// TwinCAT 3 PLC project XYZ
// ProgramVersion: 3.1.4024.0
// libraries:
//   Tc2_MC2, * (Beckhoff Automation GmbH)
//   Tc2_Standard, * (Beckhoff Automation GmbH)
//   Tc2_System, * (Beckhoff Automation GmbH)
//   Tc3_MC2_AdvancedHoming, * (Beckhoff Automation GmbH)
//   Tc3_Module, * (Beckhoff Automation GmbH)
//   Tc3_PLCopen_OpcUa, * (Beckhoff Automation GmbH)
// project tree:
//   GVLs/ GlobalSettings.TcGVL
//   / PlcTask.TcTTO
//   POUs/ FB_StorageController.TcPOU, MAIN.TcPOU, PRG_WRITE.TcPOU
// real-time tasks:
//   TASK PlcTask: cycle T#10ms, priority 20, ADS port 350
//   TASK Device 1 (OPC UA Virtual)_Task_58: cycle T#40ms, priority 58, ADS port 351
// motion (NC):
//   TASK NC-Task 1 SAF: cycle T#2ms, priority 4, ADS port 501
//   TASK NC-Task 1 SVB: cycle T#10ms, priority 8, ADS port 511
//   AXIS X1 (id 1)
//     Dynamic: Acceleration=600, Deceleration=600, Jerk=360
//     OtherSettings: AllowMotionCmdToSlave=true
//     encoder EncType=4
//       EncPara: ScaleFactorNumerator=40, ScaleFactorDenominator=12800, Inverse=true, MaxCount=#x0000ffff
//         Inc: RefSearchInverse=true, RefSyncInverse=false, RefMode=1, RefSoftSyncMask=#x0000ffff
//     drive DrvType=24
//       DrvPara: Inverse=true
//         Analog: VeloReferenz=400, ScaleFactorActTorque=0.1
//         TimeComp: TaskDelayCycles=1
//     controller CtrType=1
//       CtrPara: PriorControlFactor=1
//         Observer: BandWidth=20
//   AXIS X2 (id 2)
//     Dynamic: Acceleration=600, Deceleration=600, Jerk=360
//     OtherSettings: AllowMotionCmdToSlave=true
//     encoder EncType=4
//       EncPara: ScaleFactorNumerator=40, ScaleFactorDenominator=12800, Inverse=true, MaxCount=#x0000ffff
//         Inc: RefSearchInverse=true, RefSyncInverse=false, RefMode=1, RefSoftSyncMask=#x0000ffff
//     drive DrvType=24
//       DrvPara: Inverse=true
//         Analog: VeloReferenz=400, ScaleFactorActTorque=0.1
//         TimeComp: TaskDelayCycles=1
//     controller CtrType=1
//       CtrPara: PriorControlFactor=1
//         Observer: BandWidth=20
//   AXIS Z (id 3)
//     Dynamic: Acceleration=1.5, Deceleration=1.5, Jerk=4.5
//     Velo: Maximum=1
//     OtherSettings: AllowMotionCmdToSlave=true
//     encoder EncType=4
//       EncPara: ScaleFactorNumerator=1, ScaleFactorDenominator=12800, MaxCount=#x0000ffff
//         Inc: RefSearchInverse=true, RefSyncInverse=false, RefMode=1, RefSoftSyncMask=#x0000ffff
//     drive DrvType=24
//       Analog: VeloReferenz=1, ScaleFactorActTorque=0.1
//       TimeComp: TaskDelayCycles=1
//     controller CtrType=1
//       CtrPara: PriorControlFactor=1
//         PID: PosKp=1.5
//         Observer: BandWidth=20
//   AXIS Y (id 4)
//     OtherSettings: AllowMotionCmdToSlave=true
//     encoder EncType=4
//       EncPara: ScaleFactorNumerator=40, ScaleFactorDenominator=12800, Inverse=true, MaxCount=#x0000ffff
//         Inc: RefSearchInverse=true, RefSyncInverse=false, RefMode=1, RefSoftSyncMask=#x0000ffff
//     drive DrvType=24
//       DrvPara: Inverse=true
//         Analog: VeloReferenz=400, ScaleFactorActTorque=0.1
//         TimeComp: TaskDelayCycles=1
//     controller CtrType=1
//       CtrPara: PriorControlFactor=1
//         Observer: BandWidth=20
// I/O:
//   DEVICE Device 3 (EtherCAT) (disabled), AmsNetId 192.168.1.197.4.1
//     Term 1 (EK1100) [EK1100 EtherCAT Coupler (2A E-Bus)]
//       Term 2 (EL7031-0030) [EL7031-0030 1Ch. Stepper motor output stage (24V, 2.8A)]
//       Term 3 (EL7031-0030) [EL7031-0030 1Ch. Stepper motor output stage (24V, 2.8A)]
//       Term 4 (EL7031-0030) [EL7031-0030 1Ch. Stepper motor output stage (24V, 2.8A)]
//       Term 5 (EL7031-0030) [EL7031-0030 1Ch. Stepper motor output stage (24V, 2.8A)]
//       Term 6 (EL1008) [EL1008 8Ch. Dig. Input 24V, 3ms]
//       Term 7 (EK1110) [EK1110 EtherCAT extension]
//   DEVICE Device 1 (OPC UA Virtual), AmsNetId 192.168.1.197.2.1
// variable links:
//   NC-Task 1 SAF/Axes/X1 <-> Device 3 (EtherCAT)/Term 1 (EK1100)/Term 2 (EL7031-0030)
//     Drive/Inputs/In/nState1 @bit 3 <-> STM Status/Status/Error
//     Drive/Inputs/In/nState1 @bit 5 <-> STM Status/Status/Moving negative
//     Drive/Inputs/In/nState1 @bit 4 <-> STM Status/Status/Moving positive
//     Drive/Inputs/In/nState1 @bit 1 <-> STM Status/Status/Ready
//     Drive/Inputs/In/nState1 <-> STM Status/Status/Ready to enable
//     Drive/Inputs/In/nState1 @bit 6 <-> STM Status/Status/Torque reduced
//     Drive/Inputs/In/nState1 @bit 2 <-> STM Status/Status/Warning
//     Drive/Inputs/In/nState2 @bit 3 <-> STM Status/Status/Digital input 1
//     Drive/Inputs/In/nState2 @bit 4 <-> STM Status/Status/Digital input 2
//     Drive/Inputs/In/nState2 @bit 5 <-> STM Status/Status/Sync error
//     Drive/Inputs/In/nState2 @bit 7 <-> STM Status/Status/TxPDO Toggle
//     Drive/Inputs/In/nState4 @bit 1 <-> WcState/InputToggle
//     Drive/Inputs/In/nState4 <-> WcState/WcState
//     Drive/Outputs/Out/nCtrl1 <-> STM Control/Control/Enable
//     Drive/Outputs/Out/nCtrl1 @bit 2 <-> STM Control/Control/Reduce torque
//     Drive/Outputs/Out/nCtrl1 @bit 1 <-> STM Control/Control/Reset
//     Drive/Outputs/Out/nDataOut2[0] <-> STM Velocity/Velocity
//     Enc/Inputs/In/nDataIn1[0] <-> ENC Status compact/Counter value
//     Enc/Inputs/In/nDataIn2[0] <-> ENC Status compact/Latch value
//     Enc/Inputs/In/nState1 @bit 4 <-> ENC Status compact/Status/Counter overflow
//     Enc/Inputs/In/nState1 @bit 3 <-> ENC Status compact/Status/Counter underflow
//     Enc/Inputs/In/nState1 @bit 1 <-> ENC Status compact/Status/Latch extern valid
//     Enc/Inputs/In/nState1 @bit 2 <-> ENC Status compact/Status/Set counter done
//     Enc/Inputs/In/nState2 @bit 4 <-> ENC Status compact/Status/Status of extern latch
//     Enc/Inputs/In/nState2 @bit 5 <-> ENC Status compact/Status/Sync error
//     Enc/Inputs/In/nState2 @bit 7 <-> ENC Status compact/Status/TxPDO Toggle
//     Enc/Inputs/In/nState4 @bit 1 <-> WcState/InputToggle
//     Enc/Inputs/In/nState4 <-> WcState/WcState
//     Enc/Outputs/Out/nCtrl1 @bit 3 <-> ENC Control compact/Control/Enable latch extern on negative edge
//     Enc/Outputs/Out/nCtrl1 @bit 1 <-> ENC Control compact/Control/Enable latch extern on positive edge
//     Enc/Outputs/Out/nCtrl1 @bit 2 <-> ENC Control compact/Control/Set counter
//     Enc/Outputs/Out/nDataOut1[0] <-> ENC Control compact/Set counter value
//   NC-Task 1 SAF/Axes/X2 <-> Device 3 (EtherCAT)/Term 1 (EK1100)/Term 3 (EL7031-0030)
//     Drive/Inputs/In/nState1 @bit 3 <-> STM Status/Status/Error
//     Drive/Inputs/In/nState1 @bit 5 <-> STM Status/Status/Moving negative
//     Drive/Inputs/In/nState1 @bit 4 <-> STM Status/Status/Moving positive
//     Drive/Inputs/In/nState1 @bit 1 <-> STM Status/Status/Ready
//     Drive/Inputs/In/nState1 <-> STM Status/Status/Ready to enable
//     Drive/Inputs/In/nState1 @bit 6 <-> STM Status/Status/Torque reduced
//     Drive/Inputs/In/nState1 @bit 2 <-> STM Status/Status/Warning
//     Drive/Inputs/In/nState2 @bit 3 <-> STM Status/Status/Digital input 1
//     Drive/Inputs/In/nState2 @bit 4 <-> STM Status/Status/Digital input 2
//     Drive/Inputs/In/nState2 @bit 5 <-> STM Status/Status/Sync error
//     Drive/Inputs/In/nState2 @bit 7 <-> STM Status/Status/TxPDO Toggle
//     Drive/Inputs/In/nState4 @bit 1 <-> WcState/InputToggle
//     Drive/Inputs/In/nState4 <-> WcState/WcState
//     Drive/Outputs/Out/nCtrl1 <-> STM Control/Control/Enable
//     Drive/Outputs/Out/nCtrl1 @bit 2 <-> STM Control/Control/Reduce torque
//     Drive/Outputs/Out/nCtrl1 @bit 1 <-> STM Control/Control/Reset
//     Drive/Outputs/Out/nDataOut2[0] <-> STM Velocity/Velocity
//     Enc/Inputs/In/nDataIn1[0] <-> ENC Status compact/Counter value
//     Enc/Inputs/In/nDataIn2[0] <-> ENC Status compact/Latch value
//     Enc/Inputs/In/nState1 @bit 4 <-> ENC Status compact/Status/Counter overflow
//     Enc/Inputs/In/nState1 @bit 3 <-> ENC Status compact/Status/Counter underflow
//     Enc/Inputs/In/nState1 @bit 1 <-> ENC Status compact/Status/Latch extern valid
//     Enc/Inputs/In/nState1 @bit 2 <-> ENC Status compact/Status/Set counter done
//     Enc/Inputs/In/nState2 @bit 4 <-> ENC Status compact/Status/Status of extern latch
//     Enc/Inputs/In/nState2 @bit 5 <-> ENC Status compact/Status/Sync error
//     Enc/Inputs/In/nState2 @bit 7 <-> ENC Status compact/Status/TxPDO Toggle
//     Enc/Inputs/In/nState4 @bit 1 <-> WcState/InputToggle
//     Enc/Inputs/In/nState4 <-> WcState/WcState
//     Enc/Outputs/Out/nCtrl1 @bit 3 <-> ENC Control compact/Control/Enable latch extern on negative edge
//     Enc/Outputs/Out/nCtrl1 @bit 1 <-> ENC Control compact/Control/Enable latch extern on positive edge
//     Enc/Outputs/Out/nCtrl1 @bit 2 <-> ENC Control compact/Control/Set counter
//     Enc/Outputs/Out/nDataOut1[0] <-> ENC Control compact/Set counter value
//   NC-Task 1 SAF/Axes/Y <-> Device 3 (EtherCAT)/Term 1 (EK1100)/Term 5 (EL7031-0030)
//     Drive/Inputs/In/nState1 @bit 3 <-> STM Status/Status/Error
//     Drive/Inputs/In/nState1 @bit 5 <-> STM Status/Status/Moving negative
//     Drive/Inputs/In/nState1 @bit 4 <-> STM Status/Status/Moving positive
//     Drive/Inputs/In/nState1 @bit 1 <-> STM Status/Status/Ready
//     Drive/Inputs/In/nState1 <-> STM Status/Status/Ready to enable
//     Drive/Inputs/In/nState1 @bit 6 <-> STM Status/Status/Torque reduced
//     Drive/Inputs/In/nState1 @bit 2 <-> STM Status/Status/Warning
//     Drive/Inputs/In/nState2 @bit 3 <-> STM Status/Status/Digital input 1
//     Drive/Inputs/In/nState2 @bit 4 <-> STM Status/Status/Digital input 2
//     Drive/Inputs/In/nState2 @bit 5 <-> STM Status/Status/Sync error
//     Drive/Inputs/In/nState2 @bit 7 <-> STM Status/Status/TxPDO Toggle
//     Drive/Inputs/In/nState4 @bit 1 <-> WcState/InputToggle
//     Drive/Inputs/In/nState4 <-> WcState/WcState
//     Drive/Outputs/Out/nCtrl1 <-> STM Control/Control/Enable
//     Drive/Outputs/Out/nCtrl1 @bit 2 <-> STM Control/Control/Reduce torque
//     Drive/Outputs/Out/nCtrl1 @bit 1 <-> STM Control/Control/Reset
//     Drive/Outputs/Out/nDataOut2[0] <-> STM Velocity/Velocity
//     Enc/Inputs/In/nDataIn1[0] <-> ENC Status compact/Counter value
//     Enc/Inputs/In/nDataIn2[0] <-> ENC Status compact/Latch value
//     Enc/Inputs/In/nState1 @bit 4 <-> ENC Status compact/Status/Counter overflow
//     Enc/Inputs/In/nState1 @bit 3 <-> ENC Status compact/Status/Counter underflow
//     Enc/Inputs/In/nState1 @bit 1 <-> ENC Status compact/Status/Latch extern valid
//     Enc/Inputs/In/nState1 @bit 2 <-> ENC Status compact/Status/Set counter done
//     Enc/Inputs/In/nState2 @bit 4 <-> ENC Status compact/Status/Status of extern latch
//     Enc/Inputs/In/nState2 @bit 5 <-> ENC Status compact/Status/Sync error
//     Enc/Inputs/In/nState2 @bit 7 <-> ENC Status compact/Status/TxPDO Toggle
//     Enc/Inputs/In/nState4 @bit 1 <-> WcState/InputToggle
//     Enc/Inputs/In/nState4 <-> WcState/WcState
//     Enc/Outputs/Out/nCtrl1 @bit 3 <-> ENC Control compact/Control/Enable latch extern on negative edge
//     Enc/Outputs/Out/nCtrl1 @bit 1 <-> ENC Control compact/Control/Enable latch extern on positive edge
//     Enc/Outputs/Out/nCtrl1 @bit 2 <-> ENC Control compact/Control/Set counter
//     Enc/Outputs/Out/nDataOut1[0] <-> ENC Control compact/Set counter value
//   NC-Task 1 SAF/Axes/Z <-> Device 3 (EtherCAT)/Term 1 (EK1100)/Term 4 (EL7031-0030)
//     Drive/Inputs/In/nState1 @bit 3 <-> STM Status/Status/Error
//     Drive/Inputs/In/nState1 @bit 5 <-> STM Status/Status/Moving negative
//     Drive/Inputs/In/nState1 @bit 4 <-> STM Status/Status/Moving positive
//     Drive/Inputs/In/nState1 @bit 1 <-> STM Status/Status/Ready
//     Drive/Inputs/In/nState1 <-> STM Status/Status/Ready to enable
//     Drive/Inputs/In/nState1 @bit 6 <-> STM Status/Status/Torque reduced
//     Drive/Inputs/In/nState1 @bit 2 <-> STM Status/Status/Warning
//     Drive/Inputs/In/nState2 @bit 3 <-> STM Status/Status/Digital input 1
//     Drive/Inputs/In/nState2 @bit 4 <-> STM Status/Status/Digital input 2
//     Drive/Inputs/In/nState2 @bit 5 <-> STM Status/Status/Sync error
//     Drive/Inputs/In/nState2 @bit 7 <-> STM Status/Status/TxPDO Toggle
//     Drive/Inputs/In/nState4 @bit 1 <-> WcState/InputToggle
//     Drive/Inputs/In/nState4 <-> WcState/WcState
//     Drive/Outputs/Out/nCtrl1 <-> STM Control/Control/Enable
//     Drive/Outputs/Out/nCtrl1 @bit 2 <-> STM Control/Control/Reduce torque
//     Drive/Outputs/Out/nCtrl1 @bit 1 <-> STM Control/Control/Reset
//     Drive/Outputs/Out/nDataOut2[0] <-> STM Velocity/Velocity
//     Enc/Inputs/In/nDataIn1[0] <-> ENC Status compact/Counter value
//     Enc/Inputs/In/nDataIn2[0] <-> ENC Status compact/Latch value
//     Enc/Inputs/In/nState1 @bit 4 <-> ENC Status compact/Status/Counter overflow
//     Enc/Inputs/In/nState1 @bit 3 <-> ENC Status compact/Status/Counter underflow
//     Enc/Inputs/In/nState1 @bit 1 <-> ENC Status compact/Status/Latch extern valid
//     Enc/Inputs/In/nState1 @bit 2 <-> ENC Status compact/Status/Set counter done
//     Enc/Inputs/In/nState2 @bit 4 <-> ENC Status compact/Status/Status of extern latch
//     Enc/Inputs/In/nState2 @bit 5 <-> ENC Status compact/Status/Sync error
//     Enc/Inputs/In/nState2 @bit 7 <-> ENC Status compact/Status/TxPDO Toggle
//     Enc/Inputs/In/nState4 @bit 1 <-> WcState/InputToggle
//     Enc/Inputs/In/nState4 <-> WcState/WcState
//     Enc/Outputs/Out/nCtrl1 @bit 3 <-> ENC Control compact/Control/Enable latch extern on negative edge
//     Enc/Outputs/Out/nCtrl1 @bit 1 <-> ENC Control compact/Control/Enable latch extern on positive edge
//     Enc/Outputs/Out/nCtrl1 @bit 2 <-> ENC Control compact/Control/Set counter
//     Enc/Outputs/Out/nDataOut1[0] <-> ENC Control compact/Set counter value

CONFIGURATION XYZ
    RESOURCE PLC ON TwinCAT3
        TASK PlcTask(INTERVAL := T#10ms, PRIORITY := 20);
        PROGRAM MAIN WITH PlcTask : MAIN;
    END_RESOURCE
END_CONFIGURATION

// ---- GVLs/GlobalSettings.TcGVL
// Beckhoff Sample
VAR_GLOBAL
	sOpcUaServerUrl : STRING(MAX_STRING_LENGTH) := 'opc.tcp://PF2ADX8V:53530/OPCUA/SimulationServer'; // opc.tcp://localhost:4840 // opc.tcp://PF2ADX8V:53530/OPCUA/SimulationServer
	sNamespaceUri : STRING(MAX_STRING_LENGTH) := 'urn:PF2ADX8V:OPCUA:SimulationServer'; // TF6100 setup version 4.x default // urn:BeckhoffAutomation:Ua:PLC1 // urn:PF2ADX8V:OPCUA:SimulationServer
END_VAR

// ---- POUs/MAIN.TcPOU
PROGRAM MAIN
VAR
	// OPC/UA
	bStart : BOOL;
	fbStartTrigger : R_TRIG;
	fbConnectOPCUA : UA_Connect;
	
	// https://www.dmcinfo.com/latest-thinking/blog/id/10396/getting-started-with-opc-ua-in-beckhoff-twincat-3
	{attribute 'OPC.UA.DA' := '1'}
    hi:BOOL;
    timer: ton;
END_VAR

//PRG_WRITE();

timer(IN := NOT timer.Q, PT := T#1S) ;
IF timer.Q THEN
    hi := NOT hi;
END_IF

END_PROGRAM

// ---- POUs/FB_StorageController.TcPOU
FUNCTION_BLOCK FB_StorageController
VAR_INPUT
	bStart : BOOL; // Start the FB, power, home, ect.
	bInput : BOOL; // Set command as moving from the INPUT
	bOutput : BOOL; // Set command as moving to the OUTPUT
	bExecute : BOOL; // Start executing the current command
	nStorageLocation: BYTE; // Set command storage location
	
END_VAR
VAR_OUTPUT
	bReady : BOOL; // The FB is ready
	bBusy : BOOL; // The FB is executing a command
	bError : BOOL; // The FB is in ERROR state
	bDone : BOOL; // The FB has finished executing its command
	sError : STRING(255); // The FB ERROR description
	
END_VAR
VAR
	fbTriggerStart : R_TRIG;
	fbTriggerExecute : R_TRIG;
	
	// Axis REF
	fbAxisXa: AXIS_REF;
	fbAxisXb: AXIS_REF;
	fbAxisY:  AXIS_REF;
	fbAxisZ:  AXIS_REF;
	// Axis Power
	fbPowerXa : MC_Power;
	fbPowerXb : MC_Power;
	fbPowerY  : MC_Power;
	fbPowerZ  : MC_Power;
	// Axis Reset
	fbResetXa : MC_Reset;
	fbResetXb : MC_Reset;
	fbResetY  : MC_Reset;
	fbResetZ  : MC_Reset;
	// Axis Home
	fbHomeX : MC_Home;
	fbHomeY : MC_Home;
	fbHomeZ : MC_StepBlock;
	// Axis Gearing
	fbGearInX  : MC_GearIn;
	fbGearOutX : MC_GearOut;
	// Axis Move
	fbMoveX : MC_MoveAbsolute;
	fbMoveY : MC_MoveAbsolute;
	fbMoveZ : MC_MoveAbsolute;
	// Aixs Limit Switches
	bLimitSwitchX AT %I* : BOOL;
	bLimitSwitchY AT %I* : BOOL;
	bLimitSwitchZ AT %I* : BOOL;
	// Step Block Parameters
	fbHomeParametersZ : MC_HomingParameter;
	
	nState : BYTE;
	
END_VAR
VAR CONSTANT
	cStorageLocationCount : BYTE := 2; // The amount of storage locations
END_VAR

// Get Axis Status
fbAxisXa.ReadStatus();
fbAxisXb.ReadStatus();
fbAxisY.ReadStatus();
fbAxisZ.ReadStatus();

// Check for errors
IF bInput AND bOutput THEN
	bError := TRUE;
	sError := 'Input and Output may not be active at the same time.';
	RETURN;
END_IF

IF nStorageLocation > cStorageLocationCount THEN
	bError := TRUE;
	sError := 'Storage loacation is out of range.';
	RETURN;
END_IF

IF bExecute AND NOT bReady THEN
	bError := TRUE;
	sError := 'The FB is not ready.';
	RETURN;
END_IF

// Reset error
bError := FALSE;
sError := '';

// Get Triggers
fbTriggerStart(CLK := bStart);
fbTriggerExecute(CLK := bExecute);

// Step Through States
CASE nState OF
	000: // Idle
	fbPowerXa.Enable := FALSE;
	fbPowerXb.Enable := FALSE;
	fbPowerY.Enable := FALSE;
	fbPowerZ.Enable := FALSE;
	
	fbResetXa.Execute := FALSE;
	fbResetXb.Execute := FALSE;
	fbResetY.Execute := FALSE;
	fbResetZ.Execute := FALSE;
	
	fbHomeX.Execute := FALSE;
	fbHomeY.Execute := FALSE;
	fbHomeZ.Execute := FALSE;
	
	fbGearInX.Execute := FALSE;
	fbGearOutX.Execute := FALSE;
	
	bReady := FALSE;
	bBusy := FALSE;
	bDone := FALSE;
	
	IF fbTriggerStart.Q THEN
		bBusy := TRUE;
		nState := 010;
	END_IF
	010: // Power
	fbPowerXa.Enable := TRUE;
	fbPowerXb.Enable := TRUE;
	fbPowerY.Enable := TRUE;
	fbPowerZ.Enable := TRUE;
	
	IF fbPowerXa.Status AND fbPowerXb.Status AND fbPowerY.Status AND fbPowerZ.Status THEN nState := 020; END_IF
	020: // Couple
	IF NOT fbGearInX.InGear THEN
		fbGearInX.Execute := TRUE;
	ELSE
		nState := 030;
	END_IF
	030: // Home
	fbHomeX.Execute := TRUE;
	fbHomeY.Execute := TRUE;
	fbHomeZ.Execute := TRUE;
	
	IF fbHomeX.Done AND fbHomeY.Done AND fbHomeZ.Done THEN nState := 040; END_IF
	040: // Ready
	bReady := TRUE;
	bBusy := FALSE;
	IF fbTriggerExecute.Q THEN
		bBusy := TRUE;
		nState := 050;
	END_IF
	050: // Execute command
	// 060 -> 099 RESERVED
	100: // Move to halt possition
	110: // Decouple
	120: // Depower
	130: // Return to idle
END_CASE

fbPowerXa(Axis := fbAxisXa, Enable_Positive := TRUE, Enable_Negative := TRUE, Override := 100, BufferMode := MC_BlendingPrevious);
fbPowerXb(Axis := fbAxisXb, Enable_Positive := TRUE, Enable_Negative := TRUE, Override := 100, BufferMode := MC_BlendingPrevious);
fbPowerY(Axis := fbAxisY, Enable_Positive := TRUE, Enable_Negative := TRUE, Override := 100, BufferMode := MC_BlendingPrevious);
fbPowerZ(Axis := fbAxisZ, Enable_Positive := TRUE, Enable_Negative := TRUE, Override := 100, BufferMode := MC_BlendingPrevious);

fbResetXa(Axis := fbAxisXa);
fbResetXb(Axis := fbAxisXb);
fbResetY(Axis := fbAxisY);
fbResetZ(Axis := fbAxisZ);

fbHomeX(Axis := fbAxisXa, bCalibrationCam := bLimitSwitchX);
fbHomeY(Axis := fbAxisY, bCalibrationCam := bLimitSwitchY);
fbHomeZ(Axis := fbAxisZ, Parameter := fbHomeParametersZ);

fbGearInX(Master := fbAxisXa, Slave := fbAxisXb);
fbGearOutX(Slave := fbAxisXb);

END_FUNCTION_BLOCK

// ---- POUs/PRG_WRITE.TcPOU
// Beckhoff Sample
PROGRAM PRG_WRITE
VAR
	(* Declarations for UA_Connect *)
	fbUA_Connect			: UA_Connect;
	SessionConnectInfo		: ST_UASessionConnectInfo;
	nConnectionHdl			: DWORD;

	(* Declarations for UA_GetNamespaceIndex *)
	fbUA_GetNamespaceIndex 	: UA_GetNamespaceIndex;
	nNamespaceIndex			: UINT;

	(* Declarations for UA_NodeGetHandle *)
	fbUA_NodeGetHandle		: UA_NodeGetHandle;
	NodeID					: ST_UANodeID;
	nNodeHdl				: DWORD;

	(* Declarations for UA_Write *)
	fbUA_Write				: UA_Write;
	stIndexRange			: ARRAY [1..nMaxIndexRange] OF ST_UAIndexRange;
	nIndexRangeCount		: UINT;
	stNodeAddInfo			: ST_UANodeAdditionalInfo;
	sNodeIdentifier			: STRING(MAX_STRING_LENGTH) := 'MAIN.nNumber'; // change to node identifier
	nWriteData				: INT := 42;		// change according to the type of variable that should be written
	
	(* Declarations for UA_NodeReleaseHandle *)
	fbUA_NodeReleaseHandle	: UA_NodeReleaseHandle;

	(* Declarations for UA_Disconnect *)
	fbUA_Disconnect			: UA_Disconnect;

	(* Other declarations *)
	iState			: INT;
	bTest			: BOOL := FALSE;
	bDone			: BOOL;
	bBusy			: BOOL;
	bError			: BOOL;
	nErrorID		: DWORD;
END_VAR

// Beckhoff Sample
CASE iState OF
0:	(* idle *)
	IF bTest THEN
		bTest	:= FALSE;
		bError	:= FALSE;
		nErrorID	:= 0;

		SessionConnectInfo.tConnectTimeout 		:= T#1M;
		SessionConnectInfo.tSessionTimeout 		:= T#1M;
		SessionConnectInfo.sApplicationName		:= '';
		SessionConnectInfo.eSecurityMode 		:= eUASecurityMsgMode_None;
		SessionConnectInfo.eSecurityPolicyUri 	:= eUASecurityPolicy_None;
		SessionConnectInfo.eTransportProfileUri := eUATransportProfileUri_UATcp;

		(* Please note: when connecting to newer versions of the TwinCAT OPC UA Server,
		a server initialization is required, which basically activates username/password
		authentication for every client connection. Please set the corresponding username/password
		in stUserIdentTokenType as shown below. *)
		
		(* Please note: in order to successfully connect to the server, you need to trust the  
		server certificate. Simply move the server certificate from the "PKI\CA\rejected" to the 
		"PKI\CA\trusted" folder after the first connection. *)
 		
		(*
		SessionConnectInfo.stUserIdentTokenType.eUserIdentTokenType := eUAUITT_Username;
		SessionConnectInfo.stUserIdentTokenType.sTokenParam1 := 'Administrator';
		SessionConnectInfo.stUserIdentTokenType.sTokenParam2 := 'SomeSecurePassword';
		*)		
		
		stNodeAddInfo.nIndexRangeCount := nIndexRangeCount;
		stNodeAddInfo.stIndexRange := stIndexRange;
		iState	:= iState + 1;
	END_IF

1:	(* open UA session *)
	fbUA_Connect(
		Execute				:= TRUE,
		ServerURL			:= sOpcUaServerUrl,
		SessionConnectInfo	:= SessionConnectInfo,
		Timeout				:= T#2M,
		ConnectionHdl		=> nConnectionHdl
	);

	IF NOT fbUA_Connect.Busy THEN
		fbUA_Connect(Execute := FALSE);

		IF NOT fbUA_Connect.Error THEN
			(* session open *)
			iState := iState + 1;
		ELSE
			bError			:= TRUE;
			nErrorID		:= fbUA_Connect.ErrorID;
			nConnectionHdl	:= 0;
			iState 			:= 0; (* idle *)
		END_IF
	END_IF


2:	(* GetNS Index *)
	fbUA_GetNamespaceIndex(
		Execute			:= TRUE,
		ConnectionHdl	:= nConnectionHdl,
		NamespaceUri	:= sNamespaceUri,
		NamespaceIndex	=> nNamespaceIndex
	);

	IF NOT fbUA_GetNamespaceIndex.Busy THEN
		fbUA_GetNamespaceIndex(Execute := FALSE);

		IF NOT fbUA_GetNamespaceIndex.Error THEN
			iState 		:= iState + 1;
		ELSE
			bError		:= TRUE;
			nErrorID	:= fbUA_GetNamespaceIndex.ErrorID;
			iState 		:= 6; (* idle *)
		END_IF
	END_IF


3:	(* Get Node Handle *)
	NodeID.eIdentifierType := eUAIdentifierType_String;
	NodeID.nNamespaceIndex := nNamespaceIndex;
	NodeID.sIdentifier	:= sNodeIdentifier;
	fbUA_NodeGetHandle(
		Execute			:= TRUE,
		ConnectionHdl	:= nConnectionHdl,
		NodeID			:= NodeID,
		NodeHdl			=> nNodeHdl
	);

	IF NOT fbUA_NodeGetHandle.Busy THEN
		fbUA_NodeGetHandle(Execute := FALSE);

		IF NOT fbUA_NodeGetHandle.Error THEN
			iState 		:= iState + 1;
		ELSE
			bError		:= TRUE;
			nErrorID	:= fbUA_NodeGetHandle.ErrorID;
			iState 		:= 6; (* idle *)
		END_IF
	END_IF


4: 	(* UA_Write *)
	fbUA_Write(
		Execute			:= TRUE,
		ConnectionHdl	:= nConnectionHdl,
		NodeHdl			:= nNodeHdl,
		stNodeAddInfo	:= stNodeAddInfo,
		cbData			:= SIZEOF(nWriteData),
		pVariable		:= ADR(nWriteData)
		);

	IF NOT fbUA_Write.Busy THEN
		fbUA_Write(
			Execute 	:= FALSE,
			pVariable	:= ADR(nWriteData));

		IF NOT fbUA_Write.Error THEN
			iState 		:= iState + 1;
		ELSE
			bError		:= TRUE;
			nErrorID	:= fbUA_Write.ErrorID;
			iState 		:= 6; (* idle *)
		END_IF
	END_IF


5:	(* Release Node Handle *)
	fbUA_NodeReleaseHandle(
		Execute			:= TRUE,
		ConnectionHdl	:= nConnectionHdl,
		NodeHdl			:= nNodeHdl
	);

	IF NOT fbUA_NodeReleaseHandle.Busy THEN
		fbUA_NodeReleaseHandle(Execute := FALSE);

		IF NOT fbUA_NodeReleaseHandle.Error THEN
			iState 		:= iState + 1;
		ELSE
			bError		:= TRUE;
			nErrorID	:= fbUA_NodeReleaseHandle.ErrorID;
			iState 		:= 6; (* idle *)
		END_IF
	END_IF


6:	(* close session *)
	fbUA_Disconnect(
		Execute			:= TRUE,
		ConnectionHdl	:= nConnectionHdl
	);

	IF NOT fbUA_Disconnect.Busy THEN
		fbUA_Disconnect(Execute := FALSE);
		bBusy := FALSE; 
		IF NOT fbUA_Disconnect.Error THEN
			(* session closed *)
			iState 		:= 0;
			IF NOT bError THEN 
				bDone 	:= TRUE;
			END_IF
		ELSE
			bError			:= TRUE;
			nErrorID		:= fbUA_Disconnect.ErrorID;
			iState 			:= 0; (* idle *)
			nConnectionHdl	:= 0;
		END_IF
	END_IF
END_CASE

END_PROGRAM
